Staubli VAL3: setOpMode.pgx

public program setOpMode(num x_nAxisNum, num x_nOpMode)
  local num l_nK
begin

  //call checkDin(diSwitchedOn[x_nAxisNum],false,x_bError)

  // Interpolated position mode
  //  aioSet(aoMoop[x_nAxisNum],x_nOpMode)
  aioSet(aoWorkMode[x_nAxisNum],x_nOpMode)
  // Reset fault
//  doFaultReset[x_nAxisNum]=false
//  delay(0.1)
//  doFaultReset[x_nAxisNum]=true
//  delay(0.1)
//  doFaultReset[x_nAxisNum]=false

  // Copy current axis position into commanded position
  // Probably not necessary need to be checked.
  //  call setCmdPos(x_nAxisNum)

  //  // Init watchdog
  //  doEnableHold[x_nAxisNum]=true
  //  doWatchDog[x_nAxisNum]=true
  //  // Starting sequence
  //  doEnableVoltage[x_nAxisNum]=true
  //  doQuickStop[x_nAxisNum]=true

  //call checkDin(diReady2SwOn[x_nAxisNum],true,x_bError)


end
